TYPE ST_BWK_Parameter :
STRUCT
	Zeit_Vorl					: DINT;
	Zeit_Nachl					: DINT;

	Stellwert_Leistung_Max		: SINT;
	Stellwert_Leistung_Min		: SINT;
	Stellwert_Temperatur_Max	: SINT;
	Stellwert_Temperatur_Min	: SINT;

	Temp_Ruecklauf_Max		: REAL;
	Temp_Ruecklauf_Min		: REAL;

	AutoQuittierung			: BOOL;
END_STRUCT
END_TYPE

(* stored: Version 1.1.0.1, ProductVersion 3.1.4024.9
   DUT ST_BWK_Parameter: Id {7c70fb02-e45c-4ead-a605-418fc02b81be} *)
